TYPE E_FunctionType :
(
	eConst := 0,
	eSine,
	eSquare,
	ePulse,
	eTriangular,
	eSawtooth,
	eAM,
	eRand,
	eTrapezoid
);
END_TYPE

(* stored: Version 1.1.0.1, ProductVersion 3.1.4024.12
   DUT E_FunctionType: Id {81937273-346d-42c5-a1a3-4a9addb3025f} *)
